(* IEC 61131-3 sources: EnigmaLogic-Roomcontroller/MASTER, 3 files *)

(* ---- DisplayInterface.st ---- *)
PROGRAM DisplayInterface
VAR_EXTERNAL
DisplayAddress : usint;
DisplayAddress2 : usint;
DisplayTimeSchedule1 : int;
DisplayTimeSchedule2 : int;
DisplayTimeSchedule3 : int;
DisplayTimeSchedule4 : int;
DisplayTimeSchedule5 : int;
DisplayTemperature : real;
DisplayTemperature2 : real;
DisplayTamper : int;
DisplayPoint1 : real;
DisplayPoint2 : real;
DisplayPoint3 : real;
DisplayPoint4 : real;
DisplayPoint5 : real;
DisplayPoint6 : real;
DisplayPoint7 : real;
DisplayPoint8 : real;
DisplayPoint9 : real;
DisplayPoint10 : real;
END_VAR
VAR_GLOBAL
END_VAR
VAR
Result : int;
Result2 : real;
Resulttest : dint;
Resulttest2 : dint;
DisplayModbusMaster : ModbusRegistersFB;
SaveRegistersTimer : int := 5001;
NewValue : real;
FirstRun : int := 1;
dwTemp : dword;
diTemp : dint;

DisplayPoint2222 : real;

END_VAR

(* Read some measurements from the display *)
DisplayModbusMaster(send:=0, SlaveAddress:=DisplayAddress, StartRegister:=3000, RegisterCount:=63, RegisterType:=3, TimeOut:=200, PollInterval:=2000);
DisplayTemperature := INT_TO_REAL(WORD_TO_INT(DisplayModbusMaster.Reg0));
Result := SetRegisterF( Number := 1013, Value := REAL_TO_WORD(DisplayTemperature));

DisplayTamper := BOOL_TO_INT(DisplayModbusMaster.Reg6 = 1023);
DisplayTimeSchedule1 := WORD_TO_INT(DisplayModbusMaster.Reg7);
DisplayTimeSchedule2 := WORD_TO_INT(DisplayModbusMaster.Reg8);
DisplayTimeSchedule3 := WORD_TO_INT(DisplayModbusMaster.Reg9);
DisplayTimeSchedule4 := WORD_TO_INT(DisplayModbusMaster.Reg10);
DisplayTimeSchedule5 := WORD_TO_INT(DisplayModbusMaster.Reg11);

(* Display point overview---------------------------------------------------------------------------------------------------------- *)

(* POINT1: SET RT -> PIDHC *)

(* POINT2: ADJUST *)
DisplayPoint2 := GetDisplayPointValueF(PointNumber:=2, SlaveAddress:=DisplayAddress, OldValue:=DisplayPoint2);
Result := SetDisplayPointF(PointNumber:=2, PointType:=1, PointUnit:=0, SlaveAddress:=DisplayAddress, PointValue:=DisplayPoint2);

(* POINT3:  DO1*)
DisplayPoint3 := GetDisplayPointValueF(PointNumber:=3, SlaveAddress:=DisplayAddress, OldValue:=DisplayPoint3);
Result := SetDisplayPointF(PointNumber:=3, PointType:=0, PointUnit:=0, SlaveAddress:=DisplayAddress, PointValue:=DisplayPoint3 );
Result := SetRegisterF( Number := 12, Value := REAL_TO_WORD(DisplayPoint3));

(* POINT4:  *)
DisplayPoint4 := GetDisplayPointValueF(PointNumber:=4, SlaveAddress:=DisplayAddress, OldValue:=DisplayPoint4);
Result := SetDisplayPointF(PointNumber:=4, PointType:=0, PointUnit:=0, SlaveAddress:=DisplayAddress, PointValue:=DisplayPoint4 );

(* POINT5:  *)
DisplayPoint5 := GetDisplayPointValueF(PointNumber:=5, SlaveAddress:=DisplayAddress, OldValue:=DisplayPoint5);
Result := SetDisplayPointF(PointNumber:=5, PointType:=0, PointUnit:=0, SlaveAddress:=DisplayAddress, PointValue:=DisplayPoint5 );

(* POINT6:  *)
DisplayPoint6 := GetDisplayPointValueF(PointNumber:=6, SlaveAddress:=DisplayAddress, OldValue:=DisplayPoint6);
Result := SetDisplayPointF(PointNumber:=6, PointType:=0, PointUnit:=0, SlaveAddress:=DisplayAddress, PointValue:=DisplayPoint6 );

(* POINT7:  *)
DisplayPoint7 := GetDisplayPointValueF(PointNumber:=7, SlaveAddress:=DisplayAddress, OldValue:=DisplayPoint7);
Result := SetDisplayPointF(PointNumber:=7, PointType:=0, PointUnit:=0, SlaveAddress:=DisplayAddress, PointValue:=DisplayPoint7 );

(* POINT8: HEATING/COOLING -> PIDHC *)

(* POINT9:  *)
DisplayPoint9 := GetDisplayPointValueF(PointNumber:=9, SlaveAddress:=DisplayAddress, OldValue:=DisplayPoint9);
Result := SetDisplayPointF(PointNumber:=9, PointType:=0, PointUnit:=0, SlaveAddress:=DisplayAddress, PointValue:=DisplayPoint9 );

(* POINT10: RT -> PIDHC *)

if (DisplayTamper = 1) then
    DisplayModbusMaster.Reg62 := 0;
    DisplayModbusMaster(send:=1);
end_if;

(* Save registers if any of the setpoints is changed *)
(* 50 loop delay is to let user do all the settings before saving *)
if (SaveRegistersTimer < 50) then
    SaveRegistersTimer := SaveRegistersTimer + 1;
elsif (SaveRegistersTimer = 50) then
    SaveRegistersTimer := SaveRegistersTimer + 1;
    Result := SaveRegistersF(1);
end_if;

FirstRun:=0;
END_PROGRAM

(* ---- DISPLAYIO.ST ---- *)
PROGRAM DISPLAYIO
VAR_EXTERNAL
DisplayAddress : usint;
DisplayPoint50 : real;
DisplayPoint51 : real;
DisplayPoint52 : real;
DisplayPoint53 : real;
DisplayPoint54 : real;
DisplayPoint55 : real;
DisplayPoint56 : real;
DisplayPoint57 : real;
DisplayPoint58 : real;
DisplayPoint59 : real;
DisplayPoint60 : real;
DisplayPoint61 : real;
DisplayPoint62 : real;
DisplayPoint63 : real;
DisplayPoint64 : real;
DisplayPoint65 : real;
DisplayPoint66 : real;
DisplayPoint67 : real;
DisplayPoint68 : real;
DisplayPoint69 : real;
DisplayPoint70 : real;
DisplayPoint71 : real;
DisplayPoint72 : real;
DisplayPoint73 : real;
END_VAR

VAR_GLOBAL

END_VAR

VAR
Result : int;
Result2 : real;
END_VAR

(* Analog/Digital Input -----------------------------------------------------------------------------------------------------------*)

(* POINT50: AI1)*)
DisplayPoint50 := GetDisplayPointValueF(PointNumber:=50, SlaveAddress:=DisplayAddress, OldValue:=DisplayPoint50);
Result2 := WORD_TO_REAL(GetRegisterF(RegNumber:=500));
Result := SetDisplayPointF(PointNumber:=50, PointType:=0, PointUnit:=0, SlaveAddress:=DisplayAddress, PointValue:=Result2);

(* POINT51: AI2)*)
DisplayPoint51 := GetDisplayPointValueF(PointNumber:=51, SlaveAddress:=DisplayAddress, OldValue:=DisplayPoint51);
Result2 := WORD_TO_REAL(GetRegisterF(RegNumber:=501));
Result := SetDisplayPointF(PointNumber:=51, PointType:=0, PointUnit:=0, SlaveAddress:=DisplayAddress, PointValue:=Result2);

(* POINT52: AI3)*)
DisplayPoint52 := GetDisplayPointValueF(PointNumber:=52, SlaveAddress:=DisplayAddress, OldValue:=DisplayPoint52);
Result2 := WORD_TO_REAL(GetRegisterF(RegNumber:=502));
Result := SetDisplayPointF(PointNumber:=52, PointType:=0, PointUnit:=0, SlaveAddress:=DisplayAddress, PointValue:=Result2);

(* POINT53: AI4)*)
DisplayPoint53 := GetDisplayPointValueF(PointNumber:=53, SlaveAddress:=DisplayAddress, OldValue:=DisplayPoint53);
Result2 := WORD_TO_REAL(GetRegisterF(RegNumber:=503));
Result := SetDisplayPointF(PointNumber:=53, PointType:=0, PointUnit:=0, SlaveAddress:=DisplayAddress, PointValue:=Result2);

(* POINT54: AI5)*)
DisplayPoint54 := GetDisplayPointValueF(PointNumber:=54, SlaveAddress:=DisplayAddress, OldValue:=DisplayPoint54);
Result2 := WORD_TO_REAL(GetRegisterF(RegNumber:=504));
Result := SetDisplayPointF(PointNumber:=54, PointType:=0, PointUnit:=0, SlaveAddress:=DisplayAddress, PointValue:=Result2);

(* POINT55: AI6)*)
DisplayPoint55 := GetDisplayPointValueF(PointNumber:=55, SlaveAddress:=DisplayAddress, OldValue:=DisplayPoint55);
Result2 := WORD_TO_REAL(GetRegisterF(RegNumber:=505));
Result := SetDisplayPointF(PointNumber:=55, PointType:=0, PointUnit:=0, SlaveAddress:=DisplayAddress, PointValue:=Result2);

(* POINT56: AI7)*)
DisplayPoint56 := GetDisplayPointValueF(PointNumber:=56, SlaveAddress:=DisplayAddress, OldValue:=DisplayPoint56);
Result2 := WORD_TO_REAL(GetRegisterF(RegNumber:=506));
Result := SetDisplayPointF(PointNumber:=56, PointType:=0, PointUnit:=0, SlaveAddress:=DisplayAddress, PointValue:=Result2);

(* POINT57: AI8)*)
DisplayPoint57 := GetDisplayPointValueF(PointNumber:=57, SlaveAddress:=DisplayAddress, OldValue:=DisplayPoint57);
Result2 := WORD_TO_REAL(GetRegisterF(RegNumber:=507));
Result := SetDisplayPointF(PointNumber:=57, PointType:=0, PointUnit:=0, SlaveAddress:=DisplayAddress, PointValue:=Result2);

(* POINT58: AI9)*)
DisplayPoint58 := GetDisplayPointValueF(PointNumber:=58, SlaveAddress:=DisplayAddress, OldValue:=DisplayPoint58);
Result2 := WORD_TO_REAL(GetRegisterF(RegNumber:=508));
Result := SetDisplayPointF(PointNumber:=58, PointType:=0, PointUnit:=0, SlaveAddress:=DisplayAddress, PointValue:=Result2);

(* POINT59: AI10)*)
DisplayPoint59 := GetDisplayPointValueF(PointNumber:=59, SlaveAddress:=DisplayAddress, OldValue:=DisplayPoint59);
Result2 := WORD_TO_REAL(GetRegisterF(RegNumber:=509));
Result := SetDisplayPointF(PointNumber:=59, PointType:=0, PointUnit:=0, SlaveAddress:=DisplayAddress, PointValue:=Result2);

(* POINT60: AI11)*)
DisplayPoint60 := GetDisplayPointValueF(PointNumber:=60, SlaveAddress:=DisplayAddress, OldValue:=DisplayPoint60);
Result2 := WORD_TO_REAL(GetRegisterF(RegNumber:=510));
Result := SetDisplayPointF(PointNumber:=60, PointType:=0, PointUnit:=0, SlaveAddress:=DisplayAddress, PointValue:=Result2);

(* POINT61: AI12)*)
DisplayPoint61 := GetDisplayPointValueF(PointNumber:=61, SlaveAddress:=DisplayAddress, OldValue:=DisplayPoint61);
Result2 := WORD_TO_REAL(GetRegisterF(RegNumber:=511));
Result := SetDisplayPointF(PointNumber:=61, PointType:=0, PointUnit:=0, SlaveAddress:=DisplayAddress, PointValue:=Result2);

(* Digital Output -----------------------------------------------------------------------------------------------------------*)

(* POINT62: D01)*)
DisplayPoint62 := GetDisplayPointValueF(PointNumber:=62, SlaveAddress:=DisplayAddress, OldValue:=DisplayPoint62);
Result2 := WORD_TO_REAL(GetRegisterF(RegNumber:=12));
Result := SetDisplayPointF(PointNumber:=62, PointType:=0, PointUnit:=0, SlaveAddress:=DisplayAddress, PointValue:=Result2);

(* POINT63: D02)*)
DisplayPoint63 := GetDisplayPointValueF(PointNumber:=63, SlaveAddress:=DisplayAddress, OldValue:=DisplayPoint63);
Result2 := WORD_TO_REAL(GetRegisterF(RegNumber:=13));
Result := SetDisplayPointF(PointNumber:=63, PointType:=0, PointUnit:=0, SlaveAddress:=DisplayAddress, PointValue:=Result2);

(* POINT64: D03)*)
DisplayPoint64 := GetDisplayPointValueF(PointNumber:=64, SlaveAddress:=DisplayAddress, OldValue:=DisplayPoint64);
Result2 := WORD_TO_REAL(GetRegisterF(RegNumber:=14));
Result := SetDisplayPointF(PointNumber:=64, PointType:=0, PointUnit:=0, SlaveAddress:=DisplayAddress, PointValue:=Result2);

(* POINT65: D04)*)
DisplayPoint65 := GetDisplayPointValueF(PointNumber:=65, SlaveAddress:=DisplayAddress, OldValue:=DisplayPoint65);
Result2 := WORD_TO_REAL(GetRegisterF(RegNumber:=15));
Result := SetDisplayPointF(PointNumber:=65, PointType:=0, PointUnit:=0, SlaveAddress:=DisplayAddress, PointValue:=Result2);

(* Analog Output -----------------------------------------------------------------------------------------------------------*)

(* POINT66: A01)*)
DisplayPoint66 := GetDisplayPointValueF(PointNumber:=66, SlaveAddress:=DisplayAddress, OldValue:=DisplayPoint66);
Result2 := GetAnalogOutputF(Number:=1);
Result := SetDisplayPointF(PointNumber:=66, PointType:=0, PointUnit:=0, SlaveAddress:=DisplayAddress, PointValue:=Result2);

(* POINT67: A02)*)
DisplayPoint67 := GetDisplayPointValueF(PointNumber:=67, SlaveAddress:=DisplayAddress, OldValue:=DisplayPoint67);
Result2 := GetAnalogOutputF(Number:=2);
Result := SetDisplayPointF(PointNumber:=67, PointType:=0, PointUnit:=0, SlaveAddress:=DisplayAddress, PointValue:=Result2);

(* POINT68: A03)*)
DisplayPoint68 := GetDisplayPointValueF(PointNumber:=68, SlaveAddress:=DisplayAddress, OldValue:=DisplayPoint68);
Result2 := GetAnalogOutputF(Number:=3);
Result := SetDisplayPointF(PointNumber:=68, PointType:=0, PointUnit:=0, SlaveAddress:=DisplayAddress, PointValue:=Result2);

(* POINT69: A04)*)
DisplayPoint69 := GetDisplayPointValueF(PointNumber:=69, SlaveAddress:=DisplayAddress, OldValue:=DisplayPoint69);
Result2 := GetAnalogOutputF(Number:=4);
Result := SetDisplayPointF(PointNumber:=69, PointType:=0, PointUnit:=0, SlaveAddress:=DisplayAddress, PointValue:=Result2);

(* Triacs -----------------------------------------------------------------------------------------------------------*)

(* POINT70: T01)*)
DisplayPoint70 := GetDisplayPointValueF(PointNumber:=70, SlaveAddress:=DisplayAddress, OldValue:=DisplayPoint70);
Result2 := GetAnalogOutputF(Number:=5);
Result := SetDisplayPointF(PointNumber:=70, PointType:=0, PointUnit:=0, SlaveAddress:=DisplayAddress, PointValue:=Result2);

(* POINT71: T02)*)
DisplayPoint71 := GetDisplayPointValueF(PointNumber:=71, SlaveAddress:=DisplayAddress, OldValue:=DisplayPoint71);
Result2 := GetAnalogOutputF(Number:=6);
Result := SetDisplayPointF(PointNumber:=71, PointType:=0, PointUnit:=0, SlaveAddress:=DisplayAddress, PointValue:=Result2);

(* POINT72: T03)*)
DisplayPoint72 := GetDisplayPointValueF(PointNumber:=72, SlaveAddress:=DisplayAddress, OldValue:=DisplayPoint72);
Result2 := GetAnalogOutputF(Number:=7);
Result := SetDisplayPointF(PointNumber:=72, PointType:=0, PointUnit:=0, SlaveAddress:=DisplayAddress, PointValue:=Result2);

(* POINT73: T04)*)
DisplayPoint73 := GetDisplayPointValueF(PointNumber:=73, SlaveAddress:=DisplayAddress, OldValue:=DisplayPoint73);
Result2 := GetAnalogOutputF(Number:=8);
Result := SetDisplayPointF(PointNumber:=73, PointType:=0, PointUnit:=0, SlaveAddress:=DisplayAddress, PointValue:=Result2);
END_PROGRAM

(* ---- read_measurements.ST ---- *)
PROGRAM read_measurements
VAR
Modbus_Orja_Write : ModbusRegistersFB;
Modbus_Orja_Read : ModbusRegistersFB;
wTemp : WORD ;
temperature_word : WORD ;
Result : INT ;
dword_temp : dword ;
dword_temp2 : dword ;
dword_temp3 : dword ;
rTemp : REAL ;
DisplayPoint2 : REAL ;
Mater_relay : INT ;
Slave_relay_int : INT ;
Slave_relay_word : WORD ;
DisplayPoint1 : REAL ;
DisplayPoint3 : REAL ;
DisplayTemperature : REAL ;
FX2030_button_status : DWORD ;
FX_2030_button_pushed : BOOL ;
min01,min02,min03,min04,min05,min06,min07,min08,min09,min10,min11,min12: REAL;
END_VAR
(* set the number of register to be read and written *)
Result := SetRegisterF ( Number := 1000, Value := 9884 );

min01 := GetDisplayPointValueF(PointNumber:=1, SlaveAddress:=10, OldValue:=min01);
Result := SetRegisterF( Number := 1001, Value := REAL_TO_WORD(min01));
min02 := GetDisplayPointValueF(PointNumber:=2, SlaveAddress:=10, OldValue:=min02);
Result := SetRegisterF( Number := 1002, Value := REAL_TO_WORD(min02));
min03 := GetDisplayPointValueF(PointNumber:=3, SlaveAddress:=10, OldValue:=min03);
Result := SetRegisterF( Number := 1003, Value := REAL_TO_WORD(min03));
min04 := GetDisplayPointValueF(PointNumber:=4, SlaveAddress:=10, OldValue:=min04);
Result := SetRegisterF( Number := 1004, Value := REAL_TO_WORD(min04));
min05 := GetDisplayPointValueF(PointNumber:=5, SlaveAddress:=10, OldValue:=min05);
Result := SetRegisterF( Number := 1005, Value := REAL_TO_WORD(min05));
min06 := GetDisplayPointValueF(PointNumber:=6, SlaveAddress:=10, OldValue:=min06);
Result := SetRegisterF( Number := 1006, Value := REAL_TO_WORD(min06));
min07 := GetDisplayPointValueF(PointNumber:=7, SlaveAddress:=10, OldValue:=min07);
Result := SetRegisterF( Number := 1007, Value := REAL_TO_WORD(min07));
min08 := GetDisplayPointValueF(PointNumber:=8, SlaveAddress:=10, OldValue:=min08);
Result := SetRegisterF( Number := 1008, Value := REAL_TO_WORD(min08));
min09 := GetDisplayPointValueF(PointNumber:=9, SlaveAddress:=10, OldValue:=min09);
Result := SetRegisterF( Number := 1009, Value := REAL_TO_WORD(min09));
min10 := GetDisplayPointValueF(PointNumber:=10, SlaveAddress:=10, OldValue:=min10);
Result := SetRegisterF( Number := 1010, Value := REAL_TO_WORD(min10));
min11 := GetDisplayPointValueF(PointNumber:=11, SlaveAddress:=10, OldValue:=min11);
Result := SetRegisterF( Number := 1011, Value := REAL_TO_WORD(min11));
min12 := GetDisplayPointValueF(PointNumber:=12, SlaveAddress:=10, OldValue:=min12);
Result := SetRegisterF( Number := 1012, Value := REAL_TO_WORD(min12));

(* read the register that contains teh button status from the FX-2030 *)
FX2030_button_status := GetLongRegisterF (0) ;
FX_2030_button_pushed := INT_TO_BOOL(WORD_TO_INT(DWORD_TO_WORD(FX2030_button_status))) ;

(* read temperature from multi-24 slave module and write it to the display *)
Modbus_Orja_Read.Send := 0;
Modbus_Orja_Read.SlaveAddress := 24;
Modbus_Orja_Read.StartRegister := 523;
Modbus_Orja_Read.RegisterCount := 1;
Modbus_Orja_Read.RegisterType := 3;
Modbus_Orja_Read.TimeOut := 800;
Modbus_Orja_Read.PollInterval := 800;
Modbus_Orja_Read();
temperature_word := Modbus_Orja_Read.Reg0;
Result := word_to_int (temperature_word) ;
Result := Result / 100 ;
rTemp := INT_to_real (Result) ;

(* read button status from display and change the master multi-24 relay *)
(*
DisplayPoint2 := GetDisplayPointValueF(PointNumber:=2, SlaveAddress:=10, OldValue:=DisplayPoint2);
Mater_relay := REAL_TO_INT (DisplayPoint2) ;
*)

(* if the button on the FX-2030 is pushed, always send "0" to close the relay,
otherwise, send the status based on the button on the small display *)
(*
IF FX_2030_button_pushed THEN
	Result := SetDigitalOutputF (1, 0) ;
ELSE
	Result := SetDigitalOutputF (1, Mater_relay) ;
END_IF ;
*)
(* read button status from display and write to the slave multi-24 relay through the correct registers *)
(*
DisplayPoint3 := GetDisplayPointValueF(PointNumber:=3, SlaveAddress:=10, OldValue:=DisplayPoint3);
Slave_relay_int := REAL_TO_INT (DisplayPoint3) ;
Slave_relay_word := INT_TO_WORD (Slave_relay_int) ;
*)

(* if the button on the FX-2030 is pushed, close the relay,
otherwise, send the status based on the button on the small display *)
IF FX_2030_button_pushed THEN
	Slave_relay_word := 0 ;
END_IF ;

(* write the register to the multi-24 slave *)
Modbus_Orja_Write.Send := 1;
Modbus_Orja_Write.SlaveAddress := 24;
Modbus_Orja_Write.StartRegister := 12;
Modbus_Orja_Write.RegisterCount := 1;
Modbus_Orja_Write.RegisterType := 3;
Modbus_Orja_Write.TimeOut := 300;
Modbus_Orja_Write.PollInterval := 500;
Modbus_Orja_Write.Reg0 :=  Slave_relay_word ;
Modbus_Orja_Write();
END_PROGRAM
